// TIA Portal V19 export
TYPE "InfeedWng"
// stored: Access Published
   STRUCT
      InfeedWarning : Bool;
   END_STRUCT;
END_TYPE
